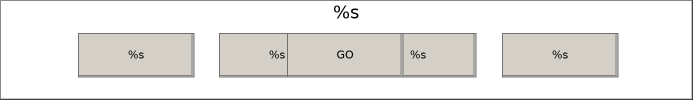
VISUALIZATION VISU_AXE_STD1_FCT_TRF_OSC  // 693x100
VAR_IN_OUT
	m_Input_MOTEUR: BLOCK_AXE_STD1_OSCILLANT;
	m_Input_PRG_MOUVEMENT_PS: BLOCK_PRG_MOUVEMENT_PS;
END_VAR
VAR_INPUT CONSTANT
	m_Input_INDEX_MOTEUR : INT;
	m_Input_Ref_Trf:		USINT;
END_VAR
    Rectangle (0,0 693x100), "%s", text list: 'TextList_Moteurs', text index: 4
    Button (78,33 116x44), "%s", text variable: m_Input_MOTEUR.CONF_ID_Poste[1], invisible if: m_Input_PRG_MOUVEMENT_PS.CONF_NB_POSTE[m_Input_INDEX_MOTEUR]<1, input disabled if: NOT m_Input_MOTEUR.OP_Position.AUTOR_IHM
        OnMouseClick: execute {
            m_Input_MOTEUR.PRM_NPOSTE:=1;
            m_Input_MOTEUR.PRM_NREF:=m_Input_REF_TRF;
            m_Input_MOTEUR.PRM_BalPos:=FALSE;
            m_Input_MOTEUR.PRM_GoToHome:=TRUE;
            m_Input_MOTEUR.PRM_Position:=0;
            m_Input_MOTEUR.OP_POSITION.ON_IHM:=TRUE;
        }
    Button (219,33 116x44), "%s", text variable: m_Input_MOTEUR.CONF_ID_Poste[2], invisible if: m_Input_PRG_MOUVEMENT_PS.CONF_NB_POSTE[m_Input_INDEX_MOTEUR]<2, input disabled if: NOT m_Input_MOTEUR.OP_Position.AUTOR_IHM
        OnMouseClick: execute {
            m_Input_MOTEUR.PRM_NPOSTE:=2;
            m_Input_MOTEUR.PRM_NREF:=m_Input_REF_TRF;
            m_Input_MOTEUR.PRM_BalPos:=FALSE;
            m_Input_MOTEUR.PRM_GoToHome:=TRUE;
            m_Input_MOTEUR.PRM_Position:=0;
            m_Input_MOTEUR.OP_POSITION.ON_IHM:=TRUE;
        }
    Button (360,33 116x44), "%s", text variable: m_Input_MOTEUR.CONF_ID_Poste[3], invisible if: m_Input_PRG_MOUVEMENT_PS.CONF_NB_POSTE[m_Input_INDEX_MOTEUR]<3, input disabled if: NOT m_Input_MOTEUR.OP_Position.AUTOR_IHM
        OnMouseClick: execute {
            m_Input_MOTEUR.PRM_NPOSTE:=3;
            m_Input_MOTEUR.PRM_NREF:=m_Input_REF_TRF;
            m_Input_MOTEUR.PRM_BalPos:=FALSE;
            m_Input_MOTEUR.PRM_GoToHome:=TRUE;
            m_Input_MOTEUR.PRM_Position:=0;
            m_Input_MOTEUR.OP_POSITION.ON_IHM:=TRUE;
        }
    Button (502,33 116x44), "%s", text variable: m_Input_MOTEUR.CONF_ID_Poste[4], invisible if: m_Input_PRG_MOUVEMENT_PS.CONF_NB_POSTE[m_Input_INDEX_MOTEUR]<4, input disabled if: NOT m_Input_MOTEUR.OP_Position.AUTOR_IHM
        OnMouseClick: execute {
            m_Input_MOTEUR.PRM_NPOSTE:=4;
            m_Input_MOTEUR.PRM_NREF:=m_Input_REF_TRF;
            m_Input_MOTEUR.PRM_BalPos:=FALSE;
            m_Input_MOTEUR.PRM_GoToHome:=TRUE;
            m_Input_MOTEUR.PRM_Position:=0;
            m_Input_MOTEUR.OP_POSITION.ON_IHM:=TRUE;
        }
    Button (287,33 116x44), "GO", invisible if: m_Input_PRG_MOUVEMENT_PS.CONF_NB_POSTE[m_Input_INDEX_MOTEUR]<>0, input disabled if: NOT m_Input_MOTEUR.OP_Position.AUTOR_IHM
        OnMouseClick: execute {
            m_Input_MOTEUR.PRM_NPOSTE:=0;
            m_Input_MOTEUR.PRM_NREF:=0;
            m_Input_MOTEUR.PRM_BalPos:=FALSE;
            m_Input_MOTEUR.PRM_GoToHome:=TRUE;
            m_Input_MOTEUR.PRM_Position:=0.0;
            m_Input_MOTEUR.OP_POSITION.ON_IHM:=TRUE;
        }
END_VISUALIZATION

(* stored: Version 1.1.0.1, ProductVersion 3.1.4024.10
   Visu VISU_AXE_STD1_FCT_TRF_OSC: Id {371fab98-e9d7-4f23-a34c-02df4120e1fd} *)
